{region '#Template'}
	{attribute 'Version' := '5.0.0.0'}
	{attribute 'Tags' := '"LCID": "1031", "Text": "Trade, Plant, Room automation"'}
	{attribute 'Tags' := '"LCID": "1033", "Text": "Trade, Plant, Room automation"'}
	{attribute 'Using' := '"Type": "Template", "URI": "Site"'}
	{attribute 'Description' := '"LCID": "1031", "Text": "Aufruf der Anlagen des Gewerks Raumautomation"'}
	{attribute 'Description' := '"LCID": "1033", "Text": "Calling the plants of the trade room automation"'}
{endregion}
FUNCTION_BLOCK FB_BA_RoomAutomation EXTENDS FB_BA_View
VAR_INPUT CONSTANT
//	RoomGeneral		: FB_BA_RoomGeneral	;
//	SampleRoom		: FB_BA_RoomSample1;			
END_VAR

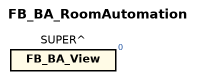
SUPER^(); // FB_BA_View

METHOD FB_init : BOOL
VAR_INPUT
	bInitRetains : BOOL; // if TRUE, the retain variables are initialized (warm start / cold start)
	bInCopyCode : BOOL;  // if TRUE, the instance afterwards gets moved into the copy code (online change)
END_VAR
//RoomGeneral.iParent			:= THIS^;
//RoomGeneral.sObjectName		:= '{RAU{Idx=01}}';
//RoomGeneral.sDescription	:= 'Room automation';
//RoomGeneral.eDPADMode		:= E_BA_DPADMode.eInclude;
//
//SampleRoom.iParent			:= THIS^;	
//SampleRoom.sObjectName		:= '{SRO{Idx=01}}';
//SampleRoom.sDescription		:= 	'Sample room'; 	
//SampleRoom.eDPADMode		:= E_BA_DPADMode.eInclude;
END_METHOD

END_FUNCTION_BLOCK

(* stored: Version 1.1.0.1, ProductVersion 3.1.4024.12
   POU FB_BA_RoomAutomation: Id {8aa4396b-0cd5-4ea5-b2b2-02d92281492e}, SpecialFunc None
   Method FB_init: Id {4b1b0a6f-5200-4809-af0e-3278ef788af7} *)
